// TIA Portal V17 export
// export: Created 2025-06-26T06:49:25.2119507Z, ExportSetting WithDefaults, DisplayName Totally Integrated Automation Portal, DisplayVersion V17 Update 8, DisplayName TIA Portal Openness, DisplayVersion V17 Update 8, DisplayName TIA Portal Version Control Interface, DisplayVersion V17, DisplayName STEP 7 Professional, DisplayVersion V17 Update 8, DisplayName STEP 7 Safety, DisplayVersion V17 Update 6, DisplayName WinCC Advanced, DisplayVersion V17 Update 8
DATA_BLOCK "DB_DO"   // DB8
{ S7_Optimized_Access := 'TRUE' }
AUTHOR : Heaten
VERSION : 0.1
// stored: AutoNumber true, DBAccessibleFromOPCUA true, DBAccessibleFromWebserver true, IsOnlyStoredInLoadMemory false, IsRetainMemResEnabled false, IsWriteProtectedInAS false, MemoryReserve 0
   VAR
      DistributionReset : Bool;   // 24V distributon control
      CabinetFan : Bool;   // PLC cabinet fan
      CabinetHeater : Bool;   // PLC cabinet heater
      HBL_EC_01 : Bool;   // Oil pan oil heaters group 1
      HBL_EC_02 : Bool;   // Oil pan oil heaters group 2
      HBL_HV_630 : Bool;   // Oil separator stage 1 oil return valve
      HBL_HV_114 : Bool;   // Suction manifold drain valve L
      HBL_HV_115 : Bool;   // Suction manifold drain valve R
      HBL_HV_860 : Bool;   // CPC tank refrigerant return selection valve
      HBL_HV_861 : Bool;   // Compressor manifold refrigerant return selection valve
      SSC_P_01 : Bool;   // SSC barrier fluid circulation pump
      SSC_F_01 : Bool;   // SSC barrier fluid cooling fan
      SSC_P_02 : Bool;   // SSC barrier fluid recharge pump
      CPC_P_01 : Bool;   // CPC refrigerant reinjection pump
      SpareContactor1 : Bool;
      SpareContactor2 : Bool;
      HBL_HV_631 : Bool;   // Oil separator stage 2 oil return valve
      HBL_HV_640_Y1 : Bool;   // Suction accumualtor drain valve open command
      HBL_HV_640_Y2 : Bool;   // Suction accumualtor drain valve close command
      HBL_HV_670_Y1 : Bool;   // Discharge accumulator drain valve open command
      HBL_HV_670_Y2 : Bool;   // Discharge accumulator drain valve close command
      CPC_HV_852_Y1 : Bool;   // CPC Cooler enable valve open command
      CPC_HV_852_Y2 : Bool;   // CPC Cooler enable valve close command
      HBL_HV_861_Y1 : Bool;   // Compressor manifold drain valve open command
      HBL_HV_861_Y2 : Bool;   // Compressor manifold drain valve close command
      HBL_HV_676 : Bool;   // Discharge accumulator drain valve 2
      HBL_HV_563 : Bool;   // Evaporator 1 axis A valve
      HBL_HV_564 : Bool;   // Evaporator 2 axis A valve
   END_VAR
BEGIN
END_DATA_BLOCK
